FUNCTION Refraction : LREAL
VAR_INPUT
	// elevation in degrees
	elevation: LREAL;
	// pressure in mBar
	pressure: LREAL := 770.0;
	// temperature in Celsius
	temperature : LREAL := 10.0;
END_VAR
VAR
END_VAR
VAR CONSTANT
	d2r:	LREAL := PI/180.0;
END_VAR

// sanity checks
elevation := LIMIT(0.0, elevation, 90.0);
pressure := LIMIT(600.0, pressure, 1200.0);
temperature := LIMIT(-30.0, temperature, 40.0);
// refraction in arcmin
Refraction := 1.02 / TAN((elevation + 10.3/(elevation + 5.11)) * d2r);
Refraction := Refraction * pressure * 283.0 / (1010.0 * (273.0 * temperature));
//refraction in degrees
Refraction := Refraction / 60.0;

END_FUNCTION

(* stored: Version 1.1.0.1, ProductVersion 3.1.4024.9
   POU Refraction: Id {064f450e-cfdd-4df5-bb63-07b8a5265b05}, SpecialFunc None *)
